// TIA Portal project "v6" (V15)

(* hardware
DEVICE "S7-1200 station_1"  S7-1200 Station
   slot 0: "Rack_0"  S7-1200 Rack  Rack  V1.0
   slot 1: "PLC_1"  CPU 1214C DC/DC/DC  6ES7 214-1AG40-0XB0  V4.2
*)

// ===== PLC "PLC_1"  CPU 1214C DC/DC/DC =====

VAR_GLOBAL   // PLC tag table "Default tag table"
   "truc1_Pulse" AT %Q0.3 : Bool;
   "truc1_Direction" AT %Q1.0 : Bool;
   "truc2_Pulse" AT %Q0.0 : Bool;
   "truc2_Direction" AT %Q0.1 : Bool;
   "truc3_Pulse" AT %Q0.4 : Bool;
   "truc3_Direction" AT %Q0.5 : Bool;
   "truc4_Pulse" AT %Q0.6 : Bool;
   "truc4_Direction" AT %Q0.7 : Bool;
   "Tag_1" AT %M0.0 : Bool;
   "Tag_2" AT %I0.0 : Bool;
   "Tag_3" AT %I0.3 : Bool;
   "vitricanden_truc1" AT %MD50 : Real;
   "kichtruc-1" AT %M1.0 : Bool;
   "Tag_6" AT %M5.0 : Bool;
   "vitricanden_truc2" AT %MD54 : Real;
   "kich_truc2" AT %M1.1 : Bool;
   "vitricanden_truc3" AT %MD58 : Real;
   "Tag_10" AT %M1.2 : Bool;
   "vitricanden_truc4" AT %MD62 : Real;
   "kich_truc4" AT %M1.3 : Bool;
   "Tag_13" AT %M5.1 : Bool;
   "Tag_14" AT %M5.2 : Bool;
   "Tag_15" AT %M5.3 : Bool;
   "Tag_16" AT %M10.0 : Bool;
   "Tag_17" AT %MW30 : Int;
   "goi vi tri" AT %M15.0 : Bool;
   "nhap vi tri goi" AT %MW32 : Int;
   "Tag_4" AT %I0.6 : Bool;
   "Tag_7" AT %I0.7 : Bool;
   "Tag_9" AT %I1.0 : Bool;
   "Tag_11" AT %I1.1 : Bool;
   "Tag_18" AT %I1.2 : Bool;
   "Tag_19" AT %I1.3 : Bool;
   "Tag_20" AT %I1.4 : Bool;
   "Tag_21" AT %I1.5 : Bool;
   "Tag_22" AT %M5.4 : Bool;
   "Tag_23" AT %M5.5 : Bool;
   "Tag_24" AT %M5.6 : Bool;
   "Tag_25" AT %M5.7 : Bool;
   "Tag_26" AT %M6.0 : Bool;
   "Tag_27" AT %M6.1 : Bool;
   "kich_truc_42" AT %M1.4 : Bool;
   "kich_truc_43" AT %M1.5 : Bool;
   "kich_truc_44" AT %M1.6 : Bool;
   "Tag_31" AT %M7.0 : Bool;
   "Tag_32" AT %M7.1 : Bool;
   "Tag_33" AT %M7.2 : Bool;
   "Tag_34" AT %M7.3 : Bool;
   "Tag_35" AT %M7.4 : Bool;
   "Tag_36" AT %M7.5 : Bool;
   "Tag_37" AT %M7.6 : Bool;
   "Tag_38" AT %M7.7 : Bool;
   "Tag_39" AT %M8.0 : Bool;
   "Tag_40" AT %M8.1 : Bool;
   "kich_truc1" AT %M2.0 : Bool;
   "kich_truc1(1)" AT %M2.1 : Bool;
   "kich_truc1(2)" AT %M2.2 : Bool;
   "kich_truc1(3)" AT %M2.3 : Bool;
   "kich_truc2(1)" AT %M2.4 : Bool;
   "kich_truc2(2)" AT %M2.5 : Bool;
   "kich_truc2(3)" AT %M2.6 : Bool;
   "kich_truc2(4)" AT %M2.7 : Bool;
   "kich_truc3(3)" AT %M3.0 : Bool;
   "kich_truc3(2)" AT %M3.1 : Bool;
   "kich_truc3" AT %M3.2 : Bool;
   "kich_truc3(1)" AT %M3.3 : Bool;
   "Tag_5" AT %M100.0 : Bool;
   "Tag_8" AT %M100.1 : Bool;
   "Tag_12" AT %M100.2 : Bool;
   "Tag_28" AT %M11.0 : Bool;
   "Tag_29" AT %M11.1 : Bool;
   "Tag_30" AT %M11.2 : Bool;
   "Tag_41" AT %M11.3 : Bool;
   "Tag_42" AT %M11.4 : Bool;
   "Tag_43" AT %M11.5 : Bool;
   "Tag_44" AT %M11.6 : Bool;
   "Tag_45" AT %M11.7 : Bool;
   "Tag_46" AT %M12.0 : Bool;
   "Tag_47" AT %M12.1 : Bool;
   "Tag_48" AT %M12.2 : Bool;
   "Tag_49" AT %M12.3 : Bool;
   "Tag_50" AT %M12.4 : Bool;
   "Tag_51" AT %M12.5 : Bool;
   "Tag_52" AT %M12.6 : Bool;
   "Tag_53" AT %M12.7 : Bool;
   "Tag_54" AT %M13.0 : Bool;
   "Tag_55" AT %M13.1 : Bool;
   "Tag_56" AT %M100.3 : Bool;
   "Tag_57" AT %M100.4 : Bool;
   "kich_truc_41" AT %M3.4 : Bool;
   "kich_truc3(4)" AT %M3.5 : Bool;
   "Kich_truc1_Home" AT %M3.6 : Bool;
   "Kich_truc2_Home" AT %M3.7 : Bool;
   "kich_truc3_Home" AT %M4.0 : Bool;
   "kich_truc4_Home" AT %M4.1 : Bool;
   "Tag_58" AT %M13.2 : Bool;
   "Tag_59" AT %M13.3 : Bool;
   "Tag_60" AT %M13.4 : Bool;
   "Tag_61" AT %M13.5 : Bool;
   "Tag_62" AT %M13.6 : Bool;
   "Tag_63" AT %M13.7 : Bool;
   "Tag_64" AT %M14.0 : Bool;
   "Tag_65" AT %M14.1 : Bool;
   "Tag_66" AT %M14.2 : Bool;
   "Tag_67" AT %M14.3 : Bool;
END_VAR

DATA_BLOCK "vitri"   // DB5
{ S7_Optimized_Access := 'FALSE' }
VERSION : 0.1
   VAR
      vitri4 : Array[0..3] of Real;
      vitri3 : Array[0..3] of Real;
      vitri2 : Array[0..3] of Real;
      Homing : Array[0..3] of Real;
      vitri1 : Array[0..3] of Real;
   END_VAR
BEGIN
END_DATA_BLOCK

DATA_BLOCK "tocdo"   // DB6
{ S7_Optimized_Access := 'FALSE' }
VERSION : 0.1
   VAR
      tocdo1 : Array[0..3] of Real;
   END_VAR
BEGIN
END_DATA_BLOCK

DATA_BLOCK "goi vitri_truc4"   // DB46
{ S7_Optimized_Access := 'TRUE' }
VERSION : 0.1
   VAR
      vitri1 : Array[0..4] of Bool;
   END_VAR
BEGIN
END_DATA_BLOCK

DATA_BLOCK "vitri_Homing"   // DB47
{ S7_Optimized_Access := 'TRUE' }
VERSION : 0.1
   VAR
      Home : Array[0..4] of Real;
   END_VAR
BEGIN
END_DATA_BLOCK

// folder: System blocks/Program resources

DATA_BLOCK "IEC_Timer_0_DB"   // DB23
{ S7_Optimized_Access := 'TRUE' }
AUTHOR : Simatic
FAMILY : IEC
NAME : IEC_TMR
VERSION : 1.0
// stored: InstanceOfName IEC_TIMER
"IEC_TIMER"
BEGIN
END_DATA_BLOCK

DATA_BLOCK "IEC_Timer_0_DB_1"   // DB24
{ S7_Optimized_Access := 'TRUE' }
AUTHOR : Simatic
FAMILY : IEC
NAME : IEC_TMR
VERSION : 1.0
// stored: InstanceOfName IEC_TIMER
"IEC_TIMER"
BEGIN
END_DATA_BLOCK

DATA_BLOCK "IEC_Timer_0_DB_2"   // DB25
{ S7_Optimized_Access := 'TRUE' }
AUTHOR : Simatic
FAMILY : IEC
NAME : IEC_TMR
VERSION : 1.0
// stored: InstanceOfName IEC_TIMER
"IEC_TIMER"
BEGIN
END_DATA_BLOCK

DATA_BLOCK "IEC_Timer_0_DB_3"   // DB26
{ S7_Optimized_Access := 'TRUE' }
AUTHOR : Simatic
FAMILY : IEC
NAME : IEC_TMR
VERSION : 1.0
// stored: InstanceOfName IEC_TIMER
"IEC_TIMER"
BEGIN
END_DATA_BLOCK

DATA_BLOCK "IEC_Timer_0_DB_4"   // DB27
{ S7_Optimized_Access := 'TRUE' }
AUTHOR : Simatic
FAMILY : IEC
NAME : IEC_TMR
VERSION : 1.0
// stored: InstanceOfName IEC_TIMER
"IEC_TIMER"
BEGIN
END_DATA_BLOCK

DATA_BLOCK "IEC_Timer_0_DB_5"   // DB28
{ S7_Optimized_Access := 'TRUE' }
AUTHOR : Simatic
FAMILY : IEC
NAME : IEC_TMR
VERSION : 1.0
// stored: InstanceOfName IEC_TIMER
"IEC_TIMER"
BEGIN
END_DATA_BLOCK

DATA_BLOCK "IEC_Timer_0_DB_6"   // DB29
{ S7_Optimized_Access := 'TRUE' }
AUTHOR : Simatic
FAMILY : IEC
NAME : IEC_TMR
VERSION : 1.0
// stored: InstanceOfName IEC_TIMER
"IEC_TIMER"
BEGIN
END_DATA_BLOCK

DATA_BLOCK "IEC_Timer_0_DB_7"   // DB30
{ S7_Optimized_Access := 'TRUE' }
AUTHOR : Simatic
FAMILY : IEC
NAME : IEC_TMR
VERSION : 1.0
// stored: InstanceOfName IEC_TIMER
"IEC_TIMER"
BEGIN
END_DATA_BLOCK

DATA_BLOCK "IEC_Timer_0_DB_8"   // DB31
{ S7_Optimized_Access := 'TRUE' }
AUTHOR : Simatic
FAMILY : IEC
NAME : IEC_TMR
VERSION : 1.0
// stored: InstanceOfName IEC_TIMER
"IEC_TIMER"
BEGIN
END_DATA_BLOCK

DATA_BLOCK "IEC_Timer_0_DB_9"   // DB32
{ S7_Optimized_Access := 'TRUE' }
AUTHOR : Simatic
FAMILY : IEC
NAME : IEC_TMR
VERSION : 1.0
// stored: InstanceOfName IEC_TIMER
"IEC_TIMER"
BEGIN
END_DATA_BLOCK

DATA_BLOCK "IEC_Timer_0_DB_10"   // DB33
{ S7_Optimized_Access := 'TRUE' }
AUTHOR : Simatic
FAMILY : IEC
NAME : IEC_TMR
VERSION : 1.0
// stored: InstanceOfName IEC_TIMER
"IEC_TIMER"
BEGIN
END_DATA_BLOCK

DATA_BLOCK "IEC_Timer_0_DB_11"   // DB34
{ S7_Optimized_Access := 'TRUE' }
AUTHOR : Simatic
FAMILY : IEC
NAME : IEC_TMR
VERSION : 1.0
// stored: InstanceOfName IEC_TIMER
"IEC_TIMER"
BEGIN
END_DATA_BLOCK

DATA_BLOCK "IEC_Timer_0_DB_12"   // DB35
{ S7_Optimized_Access := 'TRUE' }
AUTHOR : Simatic
FAMILY : IEC
NAME : IEC_TMR
VERSION : 1.0
// stored: InstanceOfName IEC_TIMER
"IEC_TIMER"
BEGIN
END_DATA_BLOCK

DATA_BLOCK "IEC_Timer_0_DB_13"   // DB36
{ S7_Optimized_Access := 'TRUE' }
AUTHOR : Simatic
FAMILY : IEC
NAME : IEC_TMR
VERSION : 1.0
// stored: InstanceOfName IEC_TIMER
"IEC_TIMER"
BEGIN
END_DATA_BLOCK

DATA_BLOCK "IEC_Timer_0_DB_14"   // DB37
{ S7_Optimized_Access := 'TRUE' }
AUTHOR : Simatic
FAMILY : IEC
NAME : IEC_TMR
VERSION : 1.0
// stored: InstanceOfName IEC_TIMER
"IEC_TIMER"
BEGIN
END_DATA_BLOCK

DATA_BLOCK "IEC_Timer_0_DB_15"   // DB38
{ S7_Optimized_Access := 'TRUE' }
AUTHOR : Simatic
FAMILY : IEC
NAME : IEC_TMR
VERSION : 1.0
// stored: InstanceOfName IEC_TIMER
"IEC_TIMER"
BEGIN
END_DATA_BLOCK

DATA_BLOCK "IEC_Timer_0_DB_16"   // DB39
{ S7_Optimized_Access := 'TRUE' }
AUTHOR : Simatic
FAMILY : IEC
NAME : IEC_TMR
VERSION : 1.0
// stored: InstanceOfName IEC_TIMER
"IEC_TIMER"
BEGIN
END_DATA_BLOCK

DATA_BLOCK "IEC_Timer_0_DB_17"   // DB40
{ S7_Optimized_Access := 'TRUE' }
AUTHOR : Simatic
FAMILY : IEC
NAME : IEC_TMR
VERSION : 1.0
// stored: InstanceOfName IEC_TIMER
"IEC_TIMER"
BEGIN
END_DATA_BLOCK

DATA_BLOCK "IEC_Timer_0_DB_18"   // DB41
{ S7_Optimized_Access := 'TRUE' }
AUTHOR : Simatic
FAMILY : IEC
NAME : IEC_TMR
VERSION : 1.0
// stored: InstanceOfName IEC_TIMER
"IEC_TIMER"
BEGIN
END_DATA_BLOCK

DATA_BLOCK "IEC_Timer_0_DB_19"   // DB42
{ S7_Optimized_Access := 'TRUE' }
AUTHOR : Simatic
FAMILY : IEC
NAME : IEC_TMR
VERSION : 1.0
// stored: InstanceOfName IEC_TIMER
"IEC_TIMER"
BEGIN
END_DATA_BLOCK

DATA_BLOCK "IEC_Timer_0_DB_20"   // DB43
{ S7_Optimized_Access := 'TRUE' }
AUTHOR : Simatic
FAMILY : IEC
NAME : IEC_TMR
VERSION : 1.0
// stored: InstanceOfName IEC_TIMER
"IEC_TIMER"
BEGIN
END_DATA_BLOCK

DATA_BLOCK "IEC_Timer_0_DB_21"   // DB44
{ S7_Optimized_Access := 'TRUE' }
AUTHOR : Simatic
FAMILY : IEC
NAME : IEC_TMR
VERSION : 1.0
// stored: InstanceOfName IEC_TIMER
"IEC_TIMER"
BEGIN
END_DATA_BLOCK

DATA_BLOCK "IEC_Timer_0_DB_22"   // DB45
{ S7_Optimized_Access := 'TRUE' }
AUTHOR : Simatic
FAMILY : IEC
NAME : IEC_TMR
VERSION : 1.0
// stored: InstanceOfName IEC_TIMER
"IEC_TIMER"
BEGIN
END_DATA_BLOCK

DATA_BLOCK "IEC_Timer_0_DB_23"   // DB48
{ S7_Optimized_Access := 'TRUE' }
AUTHOR : Simatic
FAMILY : IEC
NAME : IEC_TMR
VERSION : 1.0
// stored: InstanceOfName IEC_TIMER
"IEC_TIMER"
BEGIN
END_DATA_BLOCK

DATA_BLOCK "IEC_Timer_0_DB_24"   // DB49
{ S7_Optimized_Access := 'TRUE' }
AUTHOR : Simatic
FAMILY : IEC
NAME : IEC_TMR
VERSION : 1.0
// stored: InstanceOfName IEC_TIMER
"IEC_TIMER"
BEGIN
END_DATA_BLOCK

DATA_BLOCK "IEC_Timer_0_DB_25"   // DB50
{ S7_Optimized_Access := 'TRUE' }
AUTHOR : Simatic
FAMILY : IEC
NAME : IEC_TMR
VERSION : 1.0
// stored: InstanceOfName IEC_TIMER
"IEC_TIMER"
BEGIN
END_DATA_BLOCK

DATA_BLOCK "IEC_Timer_0_DB_26"   // DB51
{ S7_Optimized_Access := 'TRUE' }
AUTHOR : Simatic
FAMILY : IEC
NAME : IEC_TMR
VERSION : 1.0
// stored: InstanceOfName IEC_TIMER
"IEC_TIMER"
BEGIN
END_DATA_BLOCK

// folder: (top level)

DATA_BLOCK "truc1"   // DB1, Motion_DB
{ S7_Optimized_Access := 'TRUE' }
AUTHOR : SIMATIC
FAMILY : BasicMC
NAME : TO_PosAx
VERSION : 6.0
// stored: InstanceOfName TO_PositioningAxis
"TO_PositioningAxis"
BEGIN
   // Axis.DirectionOutputEnabledCU = TRUE
   // Axis.OnlinePtoModeCU = 16#0000_0002
   // Axis.SelectedChannel2EnumCU = %Q1.0
   // Axis.SelectedChannel1EnumCU = %Q0.3
   // Pulse.MinDeltaDeltaFrequencyCU = 0.004
   // Pulse.MaxDeltaDeltaFrequencyCU = 1.0E+10
   // Pulse.MinDeltaFrequencyCU = 0.005
   // Pulse.MaxDeltaFrequencyCU = 9.5E+9
   // Pulse.MinFrequencyCU = 1.0
   // Pulse.MaxFrequencyCU = 100000.0
   // Pulse.OutputSourceCU = 16#0000_0000
   // Axis.SelectPTO = 1
   // Axis.OnlinePtoIndexCU = 1
END_DATA_BLOCK

DATA_BLOCK "truc2"   // DB2, Motion_DB
{ S7_Optimized_Access := 'TRUE' }
AUTHOR : SIMATIC
FAMILY : BasicMC
NAME : TO_PosAx
VERSION : 6.0
// stored: InstanceOfName TO_PositioningAxis
"TO_PositioningAxis"
BEGIN
   // Axis.DirectionOutputEnabledCU = TRUE
   // Axis.OnlinePtoModeCU = 16#0000_0002
   // Axis.SelectedChannel2EnumCU = %Q0.1
   // Axis.SelectedChannel1EnumCU = %Q0.0
   // Pulse.MinDeltaDeltaFrequencyCU = 0.004
   // Pulse.MaxDeltaDeltaFrequencyCU = 1.0E+10
   // Pulse.MinDeltaFrequencyCU = 0.005
   // Pulse.MaxDeltaFrequencyCU = 9.5E+9
   // Pulse.MinFrequencyCU = 1.0
   // Pulse.MaxFrequencyCU = 100000.0
   // Pulse.OutputSourceCU = 16#0000_0000
   // Axis.SelectPTO = 0
END_DATA_BLOCK

DATA_BLOCK "truc3"   // DB3, Motion_DB
{ S7_Optimized_Access := 'TRUE' }
AUTHOR : SIMATIC
FAMILY : BasicMC
NAME : TO_PosAx
VERSION : 6.0
// stored: InstanceOfName TO_PositioningAxis
"TO_PositioningAxis"
BEGIN
   // Axis.DirectionOutputEnabledCU = TRUE
   // Axis.OnlinePtoModeCU = 16#0000_0002
   // Axis.SelectedChannel2EnumCU = %Q0.5
   // Axis.SelectedChannel1EnumCU = %Q0.4
   // Pulse.MinDeltaDeltaFrequencyCU = 0.004
   // Pulse.MaxDeltaDeltaFrequencyCU = 1.0E+10
   // Pulse.MinDeltaFrequencyCU = 0.005
   // Pulse.MaxDeltaFrequencyCU = 9.5E+9
   // Pulse.MinFrequencyCU = 1.0
   // Pulse.MaxFrequencyCU = 30000.0
   // Pulse.OutputSourceCU = 16#0000_0000
   // Axis.SelectPTO = 2
   // Axis.OnlinePtoIndexCU = 2
END_DATA_BLOCK

DATA_BLOCK "truc4"   // DB4, Motion_DB
{ S7_Optimized_Access := 'TRUE' }
AUTHOR : SIMATIC
FAMILY : BasicMC
NAME : TO_PosAx
VERSION : 6.0
// stored: InstanceOfName TO_PositioningAxis
"TO_PositioningAxis"
BEGIN
   // Axis.DirectionOutputEnabledCU = TRUE
   // Axis.OnlinePtoModeCU = 16#0000_0002
   // Axis.SelectedChannel2EnumCU = %Q0.7
   // Axis.SelectedChannel1EnumCU = %Q0.6
   // Pulse.MinDeltaDeltaFrequencyCU = 0.004
   // Pulse.MaxDeltaDeltaFrequencyCU = 1.0E+10
   // Pulse.MinDeltaFrequencyCU = 0.005
   // Pulse.MaxDeltaFrequencyCU = 9.5E+9
   // Pulse.MinFrequencyCU = 1.0
   // Pulse.MaxFrequencyCU = 30000.0
   // Pulse.OutputSourceCU = 16#0000_0000
   // Axis.SelectPTO = 3
   // Axis.OnlinePtoIndexCU = 3
END_DATA_BLOCK

FUNCTION "configure_initial" : Void   // FC1, LAD
{ S7_Optimized_Access := 'TRUE' }
VERSION : 0.1
BEGIN

REGION Network 1
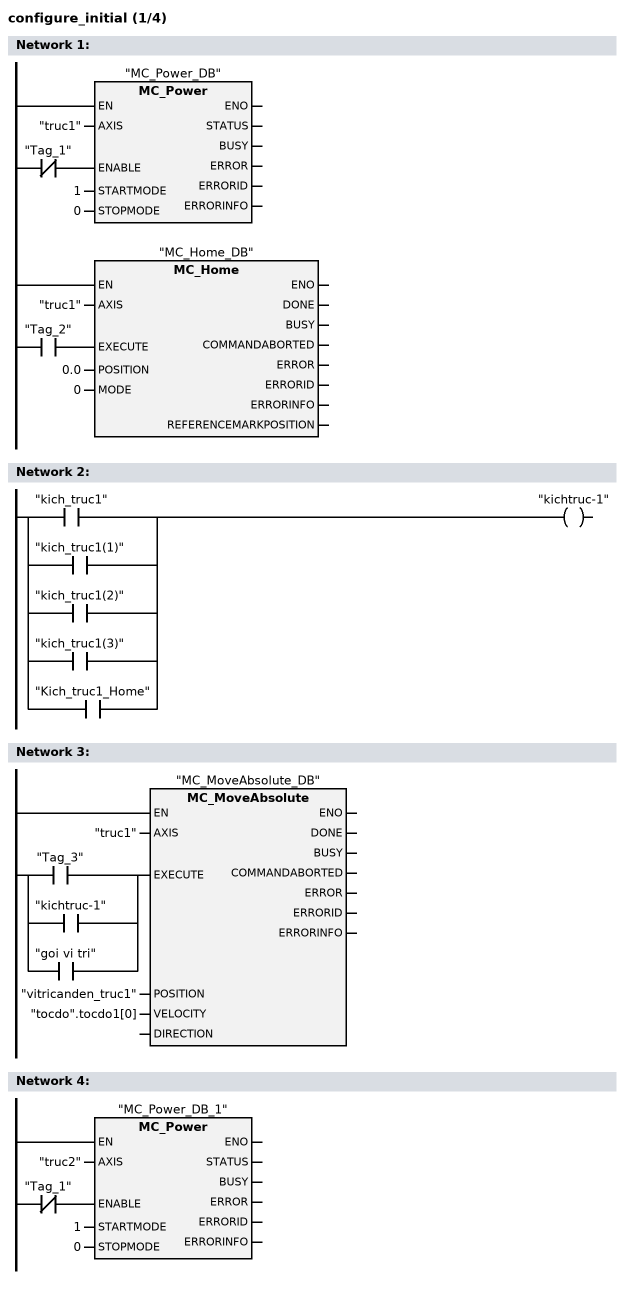
   "MC_Power_DB"(Axis := "truc1", Enable := NOT "Tag_1", StartMode := 1, StopMode := 0);   // MC_Power
   "MC_Home_DB"(Axis := "truc1", Execute := "Tag_2", Position := 0.0, Mode := 0);   // MC_Home
END_REGION

REGION Network 2
   RUNG wire#powerrail
      Contact( "kich_truc1" )
      wire#w1
      Coil( "kichtruc-1" )
   END_RUNG
   RUNG wire#powerrail
      Contact( "kich_truc1(1)" )
   END_RUNG wire#w1
   RUNG wire#powerrail
      Contact( "kich_truc1(2)" )
   END_RUNG wire#w1
   RUNG wire#powerrail
      Contact( "kich_truc1(3)" )
   END_RUNG wire#w1
   RUNG wire#powerrail
      Contact( "Kich_truc1_Home" )
   END_RUNG wire#w1
   // the same network as SCL:
   "kichtruc-1" := "kich_truc1" OR "kich_truc1(1)" OR "kich_truc1(2)" OR "kich_truc1(3)" OR "Kich_truc1_Home";
END_REGION

REGION Network 3
   "MC_MoveAbsolute_DB"(Axis := "truc1",   // MC_MoveAbsolute
                        Execute := "Tag_3" OR "kichtruc-1" OR "goi vi tri",
                        Position := "vitricanden_truc1",
                        Velocity := "tocdo".tocdo1[0]);
END_REGION

REGION Network 4
   "MC_Power_DB_1"(Axis := "truc2", Enable := NOT "Tag_1", StartMode := 1, StopMode := 0);   // MC_Power
END_REGION

REGION Network 5
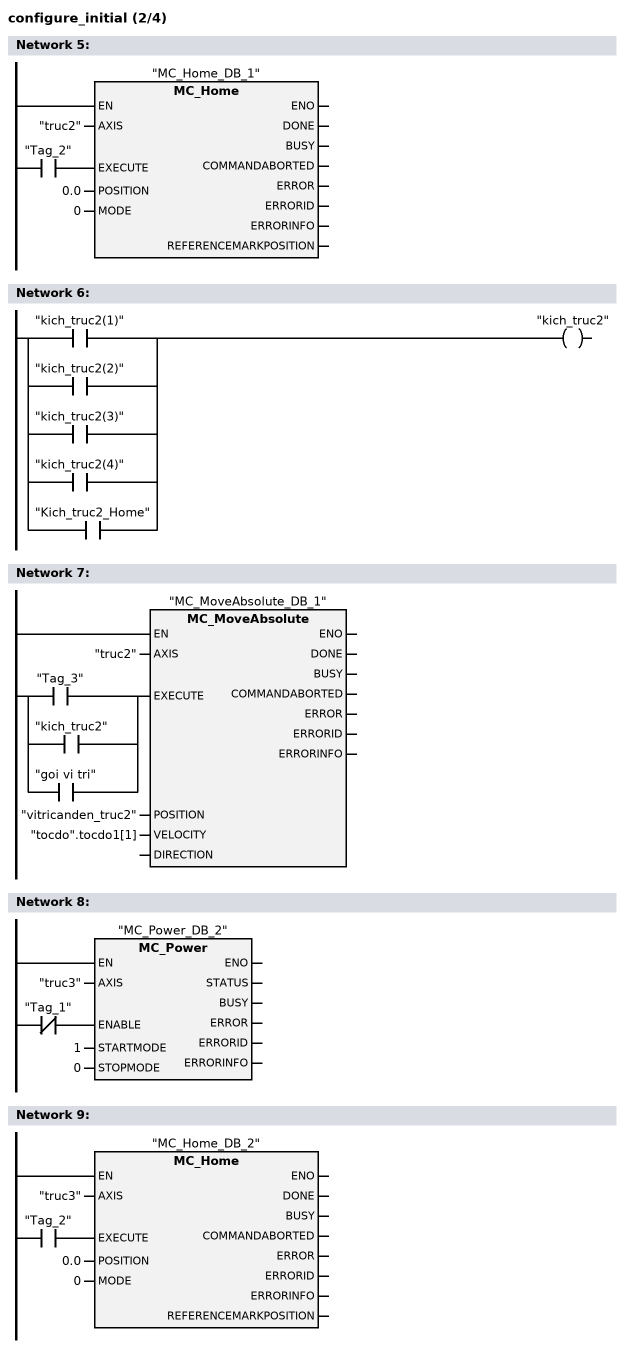
   "MC_Home_DB_1"(Axis := "truc2", Execute := "Tag_2", Position := 0.0, Mode := 0);   // MC_Home
END_REGION

REGION Network 6
   RUNG wire#powerrail
      Contact( "kich_truc2(1)" )
      wire#w1
      Coil( "kich_truc2" )
   END_RUNG
   RUNG wire#powerrail
      Contact( "kich_truc2(2)" )
   END_RUNG wire#w1
   RUNG wire#powerrail
      Contact( "kich_truc2(3)" )
   END_RUNG wire#w1
   RUNG wire#powerrail
      Contact( "kich_truc2(4)" )
   END_RUNG wire#w1
   RUNG wire#powerrail
      Contact( "Kich_truc2_Home" )
   END_RUNG wire#w1
   // the same network as SCL:
   "kich_truc2" := "kich_truc2(1)" OR "kich_truc2(2)" OR "kich_truc2(3)" OR "kich_truc2(4)" OR "Kich_truc2_Home";
END_REGION

REGION Network 7
   "MC_MoveAbsolute_DB_1"(Axis := "truc2",   // MC_MoveAbsolute
                          Execute := "Tag_3" OR "kich_truc2" OR "goi vi tri",
                          Position := "vitricanden_truc2",
                          Velocity := "tocdo".tocdo1[1]);
END_REGION

REGION Network 8
   "MC_Power_DB_2"(Axis := "truc3", Enable := NOT "Tag_1", StartMode := 1, StopMode := 0);   // MC_Power
END_REGION

REGION Network 9
   "MC_Home_DB_2"(Axis := "truc3", Execute := "Tag_2", Position := 0.0, Mode := 0);   // MC_Home
END_REGION

REGION Network 10
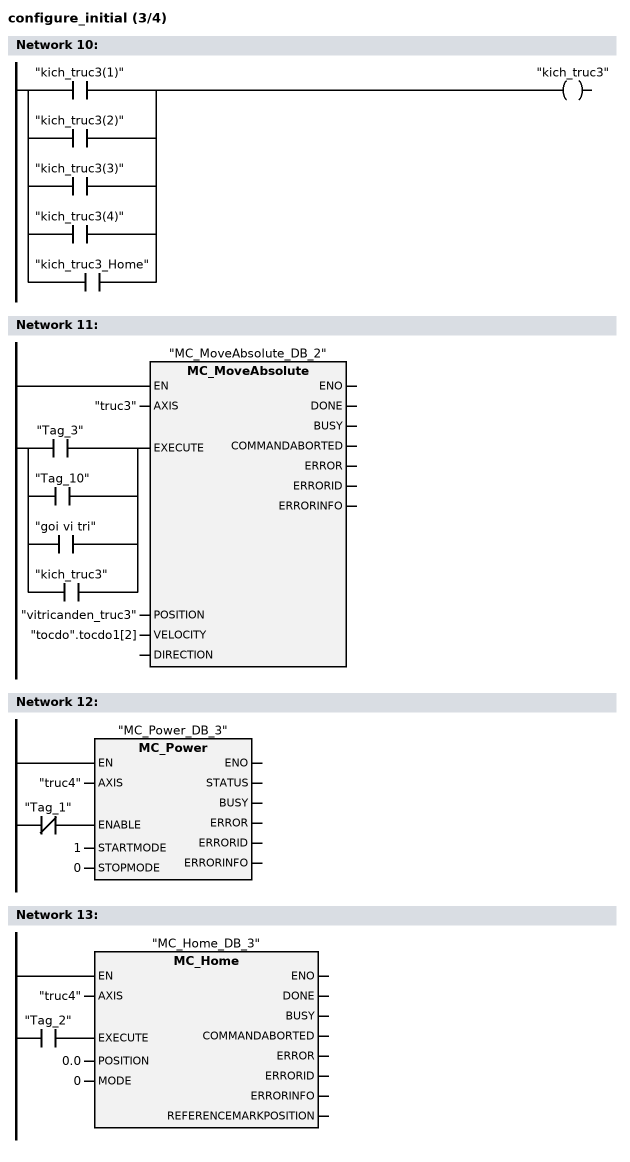
   RUNG wire#powerrail
      Contact( "kich_truc3(1)" )
      wire#w1
      Coil( "kich_truc3" )
   END_RUNG
   RUNG wire#powerrail
      Contact( "kich_truc3(2)" )
   END_RUNG wire#w1
   RUNG wire#powerrail
      Contact( "kich_truc3(3)" )
   END_RUNG wire#w1
   RUNG wire#powerrail
      Contact( "kich_truc3(4)" )
   END_RUNG wire#w1
   RUNG wire#powerrail
      Contact( "kich_truc3_Home" )
   END_RUNG wire#w1
   // the same network as SCL:
   "kich_truc3" := "kich_truc3(1)" OR "kich_truc3(2)" OR "kich_truc3(3)" OR "kich_truc3(4)" OR "kich_truc3_Home";
END_REGION

REGION Network 11
   "MC_MoveAbsolute_DB_2"(Axis := "truc3",   // MC_MoveAbsolute
                          Execute := "Tag_3" OR "Tag_10" OR "goi vi tri" OR "kich_truc3",
                          Position := "vitricanden_truc3",
                          Velocity := "tocdo".tocdo1[2]);
END_REGION

REGION Network 12
   "MC_Power_DB_3"(Axis := "truc4", Enable := NOT "Tag_1", StartMode := 1, StopMode := 0);   // MC_Power
END_REGION

REGION Network 13
   "MC_Home_DB_3"(Axis := "truc4", Execute := "Tag_2", Position := 0.0, Mode := 0);   // MC_Home
END_REGION

REGION Network 14
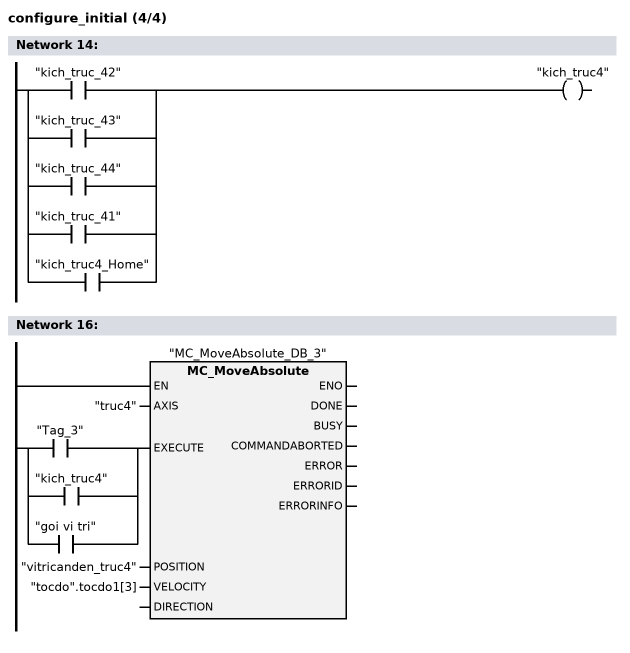
   RUNG wire#powerrail
      Contact( "kich_truc_42" )
      wire#w1
      Coil( "kich_truc4" )
   END_RUNG
   RUNG wire#powerrail
      Contact( "kich_truc_43" )
   END_RUNG wire#w1
   RUNG wire#powerrail
      Contact( "kich_truc_44" )
   END_RUNG wire#w1
   RUNG wire#powerrail
      Contact( "kich_truc_41" )
   END_RUNG wire#w1
   RUNG wire#powerrail
      Contact( "kich_truc4_Home" )
   END_RUNG wire#w1
   // the same network as SCL:
   "kich_truc4" := "kich_truc_42" OR "kich_truc_43" OR "kich_truc_44" OR "kich_truc_41" OR "kich_truc4_Home";
END_REGION

REGION Network 16
   "MC_MoveAbsolute_DB_3"(Axis := "truc4",   // MC_MoveAbsolute
                          Execute := "Tag_3" OR "kich_truc4" OR "goi vi tri",
                          Position := "vitricanden_truc4",
                          Velocity := "tocdo".tocdo1[3]);
END_REGION
END_FUNCTION

FUNCTION "luuvitri" : Void   // FC2, LAD
{ S7_Optimized_Access := 'TRUE' }
VERSION : 0.1
BEGIN

REGION Network 1
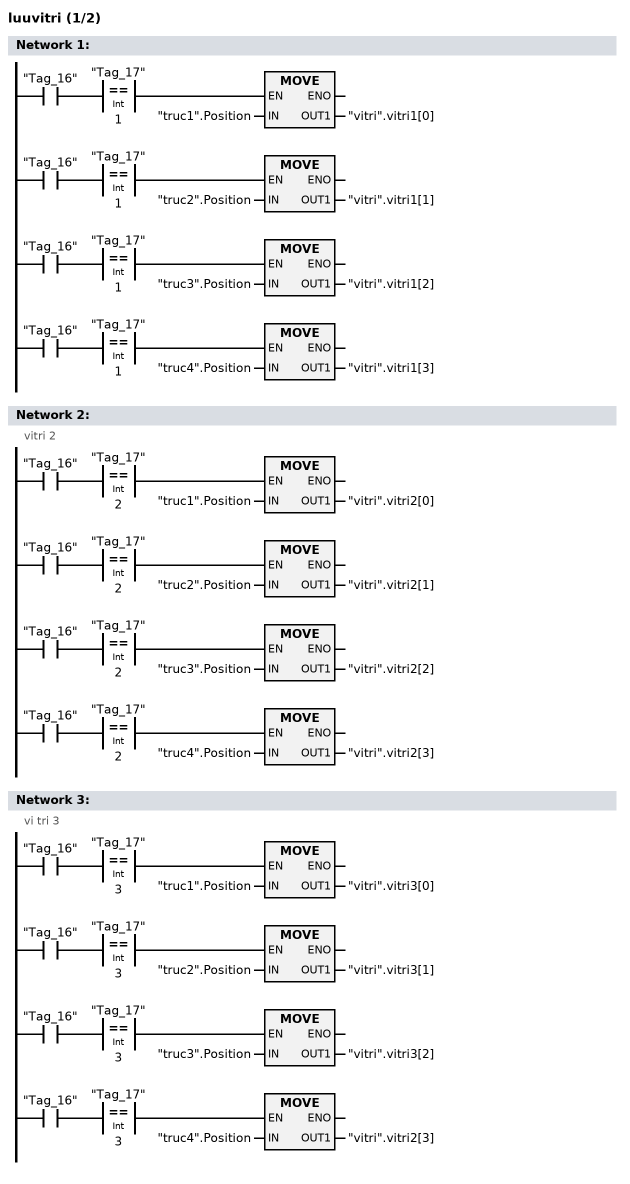
   RUNG wire#powerrail
      Contact( "Tag_16" )
      { S7_Templates := "SrcType := Int" } EQ_Contact(in1 := "Tag_17", in2 := 1)
      Move(in := "truc1".Position, out1 => "vitri".vitri1[0])
   END_RUNG
   RUNG wire#powerrail
      Contact( "Tag_16" )
      { S7_Templates := "SrcType := Int" } EQ_Contact(in1 := "Tag_17", in2 := 1)
      Move(in := "truc2".Position, out1 => "vitri".vitri1[1])
   END_RUNG
   RUNG wire#powerrail
      Contact( "Tag_16" )
      { S7_Templates := "SrcType := Int" } EQ_Contact(in1 := "Tag_17", in2 := 1)
      Move(in := "truc3".Position, out1 => "vitri".vitri1[2])
   END_RUNG
   RUNG wire#powerrail
      Contact( "Tag_16" )
      { S7_Templates := "SrcType := Int" } EQ_Contact(in1 := "Tag_17", in2 := 1)
      Move(in := "truc4".Position, out1 => "vitri".vitri1[3])
   END_RUNG
   // the same network as SCL:
   IF "Tag_16" AND ("Tag_17" = 1) THEN
       "vitri".vitri1[0] := "truc1".Position;
       "vitri".vitri1[1] := "truc2".Position;
       "vitri".vitri1[2] := "truc3".Position;
       "vitri".vitri1[3] := "truc4".Position;
   END_IF;
END_REGION

REGION Network 2
   // vitri 2
   RUNG wire#powerrail
      Contact( "Tag_16" )
      { S7_Templates := "SrcType := Int" } EQ_Contact(in1 := "Tag_17", in2 := 2)
      Move(in := "truc1".Position, out1 => "vitri".vitri2[0])
   END_RUNG
   RUNG wire#powerrail
      Contact( "Tag_16" )
      { S7_Templates := "SrcType := Int" } EQ_Contact(in1 := "Tag_17", in2 := 2)
      Move(in := "truc2".Position, out1 => "vitri".vitri2[1])
   END_RUNG
   RUNG wire#powerrail
      Contact( "Tag_16" )
      { S7_Templates := "SrcType := Int" } EQ_Contact(in1 := "Tag_17", in2 := 2)
      Move(in := "truc3".Position, out1 => "vitri".vitri2[2])
   END_RUNG
   RUNG wire#powerrail
      Contact( "Tag_16" )
      { S7_Templates := "SrcType := Int" } EQ_Contact(in1 := "Tag_17", in2 := 2)
      Move(in := "truc4".Position, out1 => "vitri".vitri2[3])
   END_RUNG
   // the same network as SCL:
   IF "Tag_16" AND ("Tag_17" = 2) THEN
       "vitri".vitri2[0] := "truc1".Position;
       "vitri".vitri2[1] := "truc2".Position;
       "vitri".vitri2[2] := "truc3".Position;
       "vitri".vitri2[3] := "truc4".Position;
   END_IF;
END_REGION

REGION Network 3
   // vi tri 3
   RUNG wire#powerrail
      Contact( "Tag_16" )
      { S7_Templates := "SrcType := Int" } EQ_Contact(in1 := "Tag_17", in2 := 3)
      Move(in := "truc1".Position, out1 => "vitri".vitri3[0])
   END_RUNG
   RUNG wire#powerrail
      Contact( "Tag_16" )
      { S7_Templates := "SrcType := Int" } EQ_Contact(in1 := "Tag_17", in2 := 3)
      Move(in := "truc2".Position, out1 => "vitri".vitri3[1])
   END_RUNG
   RUNG wire#powerrail
      Contact( "Tag_16" )
      { S7_Templates := "SrcType := Int" } EQ_Contact(in1 := "Tag_17", in2 := 3)
      Move(in := "truc3".Position, out1 => "vitri".vitri3[2])
   END_RUNG
   RUNG wire#powerrail
      Contact( "Tag_16" )
      { S7_Templates := "SrcType := Int" } EQ_Contact(in1 := "Tag_17", in2 := 3)
      Move(in := "truc4".Position, out1 => "vitri".vitri2[3])
   END_RUNG
   // the same network as SCL:
   IF "Tag_16" AND ("Tag_17" = 3) THEN
       "vitri".vitri3[0] := "truc1".Position;
       "vitri".vitri3[1] := "truc2".Position;
       "vitri".vitri3[2] := "truc3".Position;
       "vitri".vitri2[3] := "truc4".Position;
   END_IF;
END_REGION

REGION Network 4
   // vi tri 3
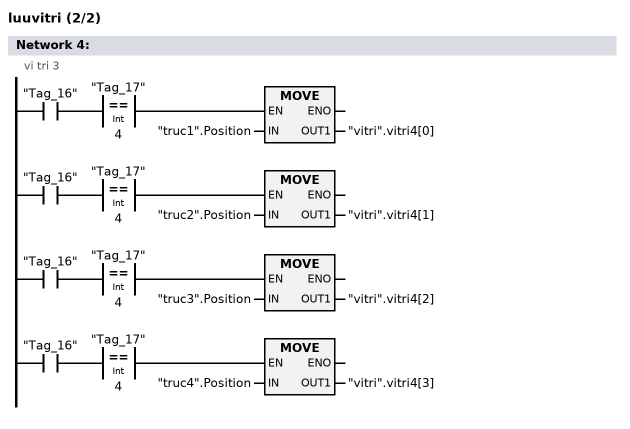
   RUNG wire#powerrail
      Contact( "Tag_16" )
      { S7_Templates := "SrcType := Int" } EQ_Contact(in1 := "Tag_17", in2 := 4)
      Move(in := "truc1".Position, out1 => "vitri".vitri4[0])
   END_RUNG
   RUNG wire#powerrail
      Contact( "Tag_16" )
      { S7_Templates := "SrcType := Int" } EQ_Contact(in1 := "Tag_17", in2 := 4)
      Move(in := "truc2".Position, out1 => "vitri".vitri4[1])
   END_RUNG
   RUNG wire#powerrail
      Contact( "Tag_16" )
      { S7_Templates := "SrcType := Int" } EQ_Contact(in1 := "Tag_17", in2 := 4)
      Move(in := "truc3".Position, out1 => "vitri".vitri4[2])
   END_RUNG
   RUNG wire#powerrail
      Contact( "Tag_16" )
      { S7_Templates := "SrcType := Int" } EQ_Contact(in1 := "Tag_17", in2 := 4)
      Move(in := "truc4".Position, out1 => "vitri".vitri4[3])
   END_RUNG
   // the same network as SCL:
   IF "Tag_16" AND ("Tag_17" = 4) THEN
       "vitri".vitri4[0] := "truc1".Position;
       "vitri".vitri4[1] := "truc2".Position;
       "vitri".vitri4[2] := "truc3".Position;
       "vitri".vitri4[3] := "truc4".Position;
   END_IF;
END_REGION
END_FUNCTION

FUNCTION "goivitri" : Void   // FC3, LAD
{ S7_Optimized_Access := 'TRUE' }
VERSION : 0.1
BEGIN

REGION Network 1
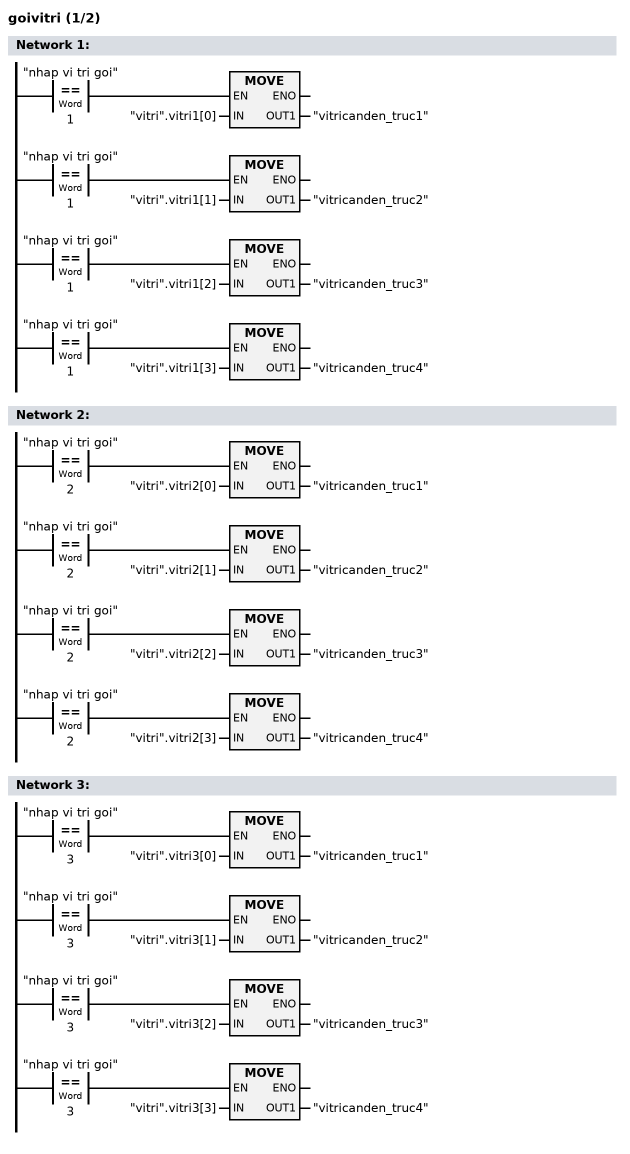
   RUNG wire#powerrail
      { S7_Templates := "SrcType := Word" } EQ_Contact(in1 := "nhap vi tri goi", in2 := 1)
      Move(in := "vitri".vitri1[0], out1 => "vitricanden_truc1")
   END_RUNG
   RUNG wire#powerrail
      { S7_Templates := "SrcType := Word" } EQ_Contact(in1 := "nhap vi tri goi", in2 := 1)
      Move(in := "vitri".vitri1[1], out1 => "vitricanden_truc2")
   END_RUNG
   RUNG wire#powerrail
      { S7_Templates := "SrcType := Word" } EQ_Contact(in1 := "nhap vi tri goi", in2 := 1)
      Move(in := "vitri".vitri1[2], out1 => "vitricanden_truc3")
   END_RUNG
   RUNG wire#powerrail
      { S7_Templates := "SrcType := Word" } EQ_Contact(in1 := "nhap vi tri goi", in2 := 1)
      Move(in := "vitri".vitri1[3], out1 => "vitricanden_truc4")
   END_RUNG
   // the same network as SCL:
   IF "nhap vi tri goi" = 1 THEN
       "vitricanden_truc1" := "vitri".vitri1[0];
       "vitricanden_truc2" := "vitri".vitri1[1];
       "vitricanden_truc3" := "vitri".vitri1[2];
       "vitricanden_truc4" := "vitri".vitri1[3];
   END_IF;
END_REGION

REGION Network 2
   RUNG wire#powerrail
      { S7_Templates := "SrcType := Word" } EQ_Contact(in1 := "nhap vi tri goi", in2 := 2)
      Move(in := "vitri".vitri2[0], out1 => "vitricanden_truc1")
   END_RUNG
   RUNG wire#powerrail
      { S7_Templates := "SrcType := Word" } EQ_Contact(in1 := "nhap vi tri goi", in2 := 2)
      Move(in := "vitri".vitri2[1], out1 => "vitricanden_truc2")
   END_RUNG
   RUNG wire#powerrail
      { S7_Templates := "SrcType := Word" } EQ_Contact(in1 := "nhap vi tri goi", in2 := 2)
      Move(in := "vitri".vitri2[2], out1 => "vitricanden_truc3")
   END_RUNG
   RUNG wire#powerrail
      { S7_Templates := "SrcType := Word" } EQ_Contact(in1 := "nhap vi tri goi", in2 := 2)
      Move(in := "vitri".vitri2[3], out1 => "vitricanden_truc4")
   END_RUNG
   // the same network as SCL:
   IF "nhap vi tri goi" = 2 THEN
       "vitricanden_truc1" := "vitri".vitri2[0];
       "vitricanden_truc2" := "vitri".vitri2[1];
       "vitricanden_truc3" := "vitri".vitri2[2];
       "vitricanden_truc4" := "vitri".vitri2[3];
   END_IF;
END_REGION

REGION Network 3
   RUNG wire#powerrail
      { S7_Templates := "SrcType := Word" } EQ_Contact(in1 := "nhap vi tri goi", in2 := 3)
      Move(in := "vitri".vitri3[0], out1 => "vitricanden_truc1")
   END_RUNG
   RUNG wire#powerrail
      { S7_Templates := "SrcType := Word" } EQ_Contact(in1 := "nhap vi tri goi", in2 := 3)
      Move(in := "vitri".vitri3[1], out1 => "vitricanden_truc2")
   END_RUNG
   RUNG wire#powerrail
      { S7_Templates := "SrcType := Word" } EQ_Contact(in1 := "nhap vi tri goi", in2 := 3)
      Move(in := "vitri".vitri3[2], out1 => "vitricanden_truc3")
   END_RUNG
   RUNG wire#powerrail
      { S7_Templates := "SrcType := Word" } EQ_Contact(in1 := "nhap vi tri goi", in2 := 3)
      Move(in := "vitri".vitri3[3], out1 => "vitricanden_truc4")
   END_RUNG
   // the same network as SCL:
   IF "nhap vi tri goi" = 3 THEN
       "vitricanden_truc1" := "vitri".vitri3[0];
       "vitricanden_truc2" := "vitri".vitri3[1];
       "vitricanden_truc3" := "vitri".vitri3[2];
       "vitricanden_truc4" := "vitri".vitri3[3];
   END_IF;
END_REGION

REGION Network 4
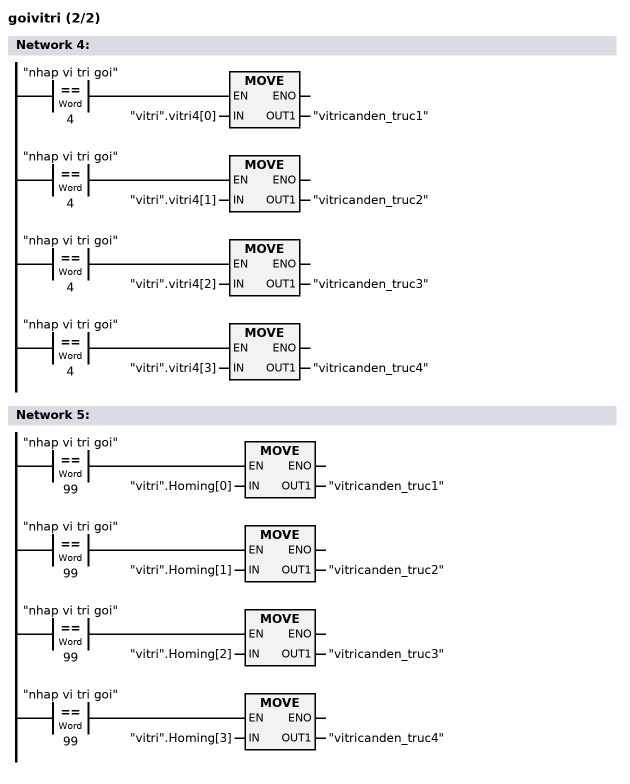
   RUNG wire#powerrail
      { S7_Templates := "SrcType := Word" } EQ_Contact(in1 := "nhap vi tri goi", in2 := 4)
      Move(in := "vitri".vitri4[0], out1 => "vitricanden_truc1")
   END_RUNG
   RUNG wire#powerrail
      { S7_Templates := "SrcType := Word" } EQ_Contact(in1 := "nhap vi tri goi", in2 := 4)
      Move(in := "vitri".vitri4[1], out1 => "vitricanden_truc2")
   END_RUNG
   RUNG wire#powerrail
      { S7_Templates := "SrcType := Word" } EQ_Contact(in1 := "nhap vi tri goi", in2 := 4)
      Move(in := "vitri".vitri4[2], out1 => "vitricanden_truc3")
   END_RUNG
   RUNG wire#powerrail
      { S7_Templates := "SrcType := Word" } EQ_Contact(in1 := "nhap vi tri goi", in2 := 4)
      Move(in := "vitri".vitri4[3], out1 => "vitricanden_truc4")
   END_RUNG
   // the same network as SCL:
   IF "nhap vi tri goi" = 4 THEN
       "vitricanden_truc1" := "vitri".vitri4[0];
       "vitricanden_truc2" := "vitri".vitri4[1];
       "vitricanden_truc3" := "vitri".vitri4[2];
       "vitricanden_truc4" := "vitri".vitri4[3];
   END_IF;
END_REGION

REGION Network 5
   RUNG wire#powerrail
      { S7_Templates := "SrcType := Word" } EQ_Contact(in1 := "nhap vi tri goi", in2 := 99)
      Move(in := "vitri".Homing[0], out1 => "vitricanden_truc1")
   END_RUNG
   RUNG wire#powerrail
      { S7_Templates := "SrcType := Word" } EQ_Contact(in1 := "nhap vi tri goi", in2 := 99)
      Move(in := "vitri".Homing[1], out1 => "vitricanden_truc2")
   END_RUNG
   RUNG wire#powerrail
      { S7_Templates := "SrcType := Word" } EQ_Contact(in1 := "nhap vi tri goi", in2 := 99)
      Move(in := "vitri".Homing[2], out1 => "vitricanden_truc3")
   END_RUNG
   RUNG wire#powerrail
      { S7_Templates := "SrcType := Word" } EQ_Contact(in1 := "nhap vi tri goi", in2 := 99)
      Move(in := "vitri".Homing[3], out1 => "vitricanden_truc4")
   END_RUNG
   // the same network as SCL:
   IF "nhap vi tri goi" = 99 THEN
       "vitricanden_truc1" := "vitri".Homing[0];
       "vitricanden_truc2" := "vitri".Homing[1];
       "vitricanden_truc3" := "vitri".Homing[2];
       "vitricanden_truc4" := "vitri".Homing[3];
   END_IF;
END_REGION
END_FUNCTION

FUNCTION "Run_Job" : Void   // FC4, LAD
{ S7_Optimized_Access := 'TRUE' }
VERSION : 0.1
BEGIN

REGION Network 1
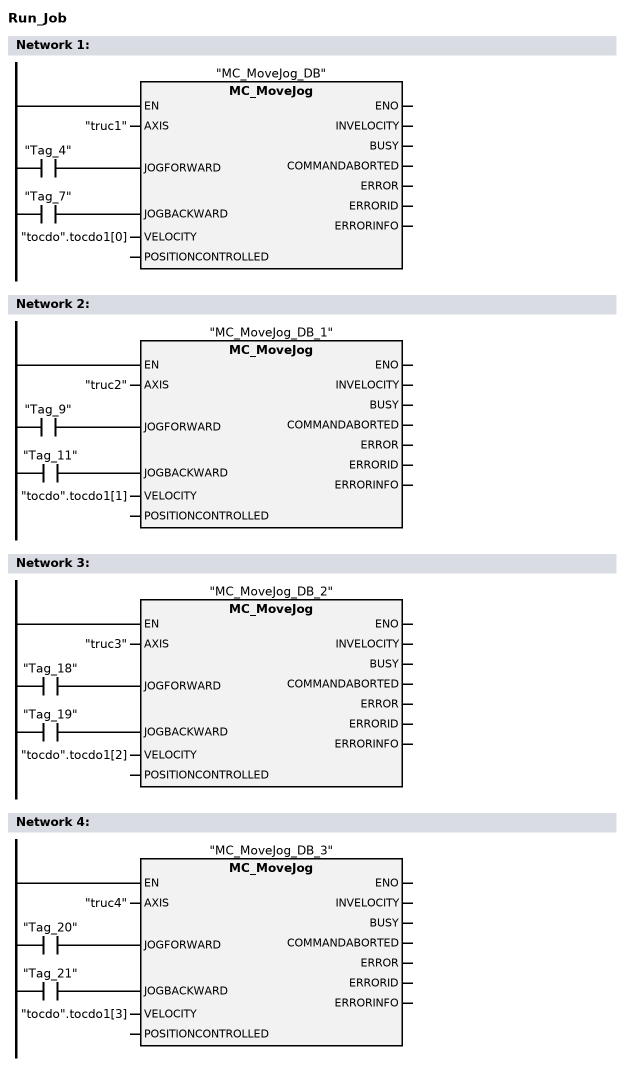
   "MC_MoveJog_DB"(Axis := "truc1",   // MC_MoveJog
                   JogForward := "Tag_4",
                   JogBackward := "Tag_7",
                   Velocity := "tocdo".tocdo1[0]);
END_REGION

REGION Network 2
   "MC_MoveJog_DB_1"(Axis := "truc2",   // MC_MoveJog
                     JogForward := "Tag_9",
                     JogBackward := "Tag_11",
                     Velocity := "tocdo".tocdo1[1]);
END_REGION

REGION Network 3
   "MC_MoveJog_DB_2"(Axis := "truc3",   // MC_MoveJog
                     JogForward := "Tag_18",
                     JogBackward := "Tag_19",
                     Velocity := "tocdo".tocdo1[2]);
END_REGION

REGION Network 4
   "MC_MoveJog_DB_3"(Axis := "truc4",   // MC_MoveJog
                     JogForward := "Tag_20",
                     JogBackward := "Tag_21",
                     Velocity := "tocdo".tocdo1[3]);
END_REGION
END_FUNCTION

FUNCTION "BT_Giua_Khau1" : Void   // FC5, LAD
{ S7_Optimized_Access := 'TRUE' }
VERSION : 0.1
BEGIN

REGION Network 1
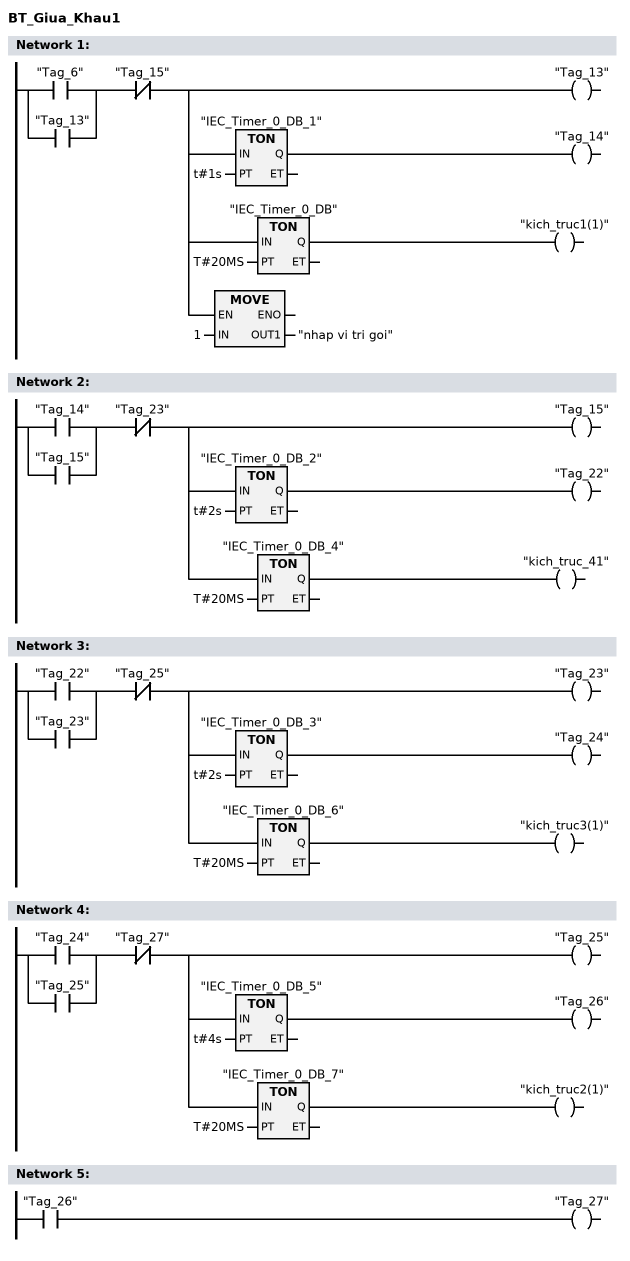
   "Tag_13" := ("Tag_6" OR "Tag_13") AND NOT "Tag_15";
   "IEC_Timer_0_DB_1".TON(IN := "Tag_13", PT := t#1s);
   "Tag_14" := "IEC_Timer_0_DB_1".Q;
   "IEC_Timer_0_DB".TON(IN := "Tag_13", PT := T#20MS);
   "kich_truc1(1)" := "IEC_Timer_0_DB".Q;
   IF "Tag_13" THEN "nhap vi tri goi" := 1; END_IF;
END_REGION

REGION Network 2
   "Tag_15" := ("Tag_14" OR "Tag_15") AND NOT "Tag_23";
   "IEC_Timer_0_DB_2".TON(IN := "Tag_15", PT := t#2s);
   "Tag_22" := "IEC_Timer_0_DB_2".Q;
   "IEC_Timer_0_DB_4".TON(IN := "Tag_15", PT := T#20MS);
   "kich_truc_41" := "IEC_Timer_0_DB_4".Q;
END_REGION

REGION Network 3
   "Tag_23" := ("Tag_22" OR "Tag_23") AND NOT "Tag_25";
   "IEC_Timer_0_DB_3".TON(IN := "Tag_23", PT := t#2s);
   "Tag_24" := "IEC_Timer_0_DB_3".Q;
   "IEC_Timer_0_DB_6".TON(IN := "Tag_23", PT := T#20MS);
   "kich_truc3(1)" := "IEC_Timer_0_DB_6".Q;
END_REGION

REGION Network 4
   "Tag_25" := ("Tag_24" OR "Tag_25") AND NOT "Tag_27";
   "IEC_Timer_0_DB_5".TON(IN := "Tag_25", PT := t#4s);
   "Tag_26" := "IEC_Timer_0_DB_5".Q;
   "IEC_Timer_0_DB_7".TON(IN := "Tag_25", PT := T#20MS);
   "kich_truc2(1)" := "IEC_Timer_0_DB_7".Q;
END_REGION

REGION Network 5
   RUNG wire#powerrail
      Contact( "Tag_26" )
      Coil( "Tag_27" )
   END_RUNG
   // the same network as SCL:
   "Tag_27" := "Tag_26";
END_REGION
END_FUNCTION

FUNCTION "BT_Giua_Khau2" : Void   // FC6, LAD
{ S7_Optimized_Access := 'TRUE' }
VERSION : 0.1
BEGIN

REGION Network 1
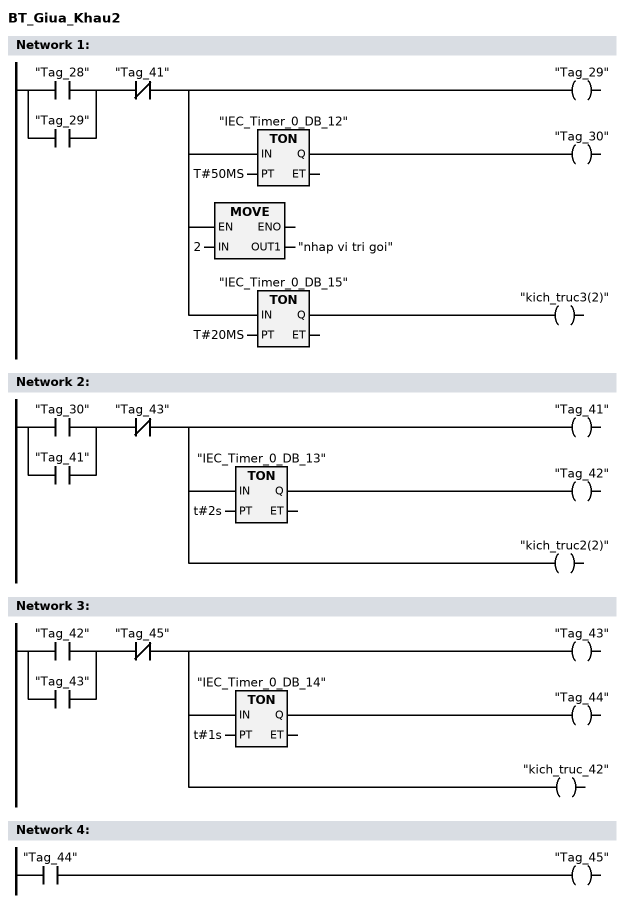
   "Tag_29" := ("Tag_28" OR "Tag_29") AND NOT "Tag_41";
   "IEC_Timer_0_DB_12".TON(IN := "Tag_29", PT := T#50MS);
   "Tag_30" := "IEC_Timer_0_DB_12".Q;
   IF "Tag_29" THEN "nhap vi tri goi" := 2; END_IF;
   "IEC_Timer_0_DB_15".TON(IN := "Tag_29", PT := T#20MS);
   "kich_truc3(2)" := "IEC_Timer_0_DB_15".Q;
END_REGION

REGION Network 2
   "Tag_41" := ("Tag_30" OR "Tag_41") AND NOT "Tag_43";
   "IEC_Timer_0_DB_13".TON(IN := "Tag_41", PT := t#2s);
   "Tag_42" := "IEC_Timer_0_DB_13".Q;
   "kich_truc2(2)" := "Tag_41";
END_REGION

REGION Network 3
   "Tag_43" := ("Tag_42" OR "Tag_43") AND NOT "Tag_45";
   "IEC_Timer_0_DB_14".TON(IN := "Tag_43", PT := t#1s);
   "Tag_44" := "IEC_Timer_0_DB_14".Q;
   "kich_truc_42" := "Tag_43";
END_REGION

REGION Network 4
   RUNG wire#powerrail
      Contact( "Tag_44" )
      Coil( "Tag_45" )
   END_RUNG
   // the same network as SCL:
   "Tag_45" := "Tag_44";
END_REGION
END_FUNCTION

FUNCTION "BT_Giua_khau3" : Void   // FC7, LAD
{ S7_Optimized_Access := 'TRUE' }
VERSION : 0.1
BEGIN

REGION Network 1
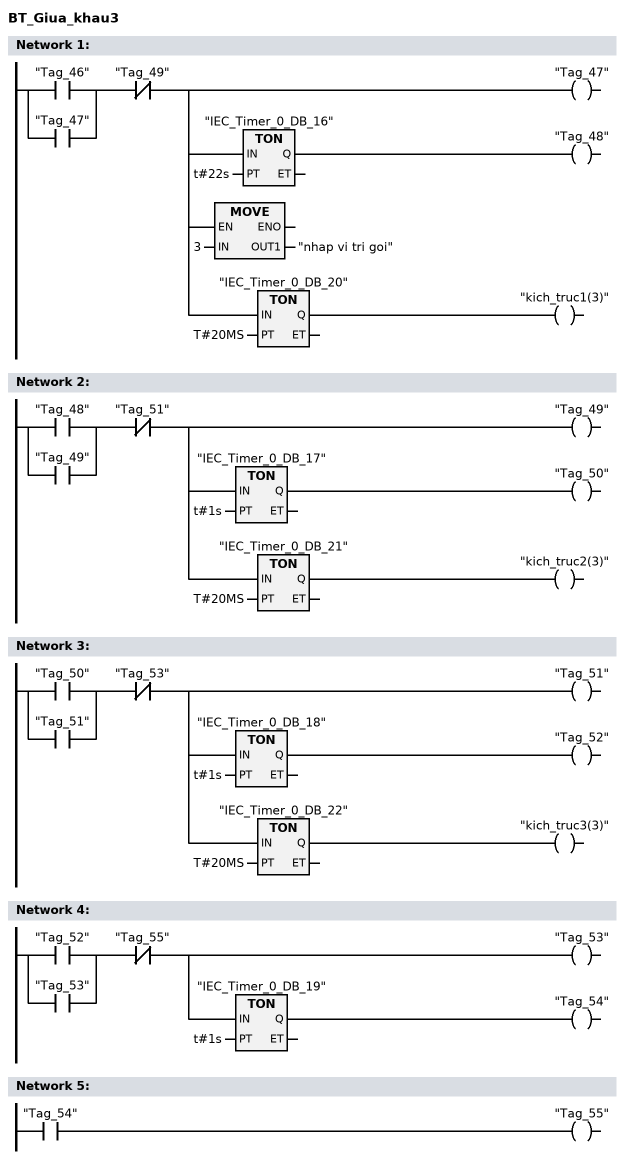
   "Tag_47" := ("Tag_46" OR "Tag_47") AND NOT "Tag_49";
   "IEC_Timer_0_DB_16".TON(IN := "Tag_47", PT := t#22s);
   "Tag_48" := "IEC_Timer_0_DB_16".Q;
   IF "Tag_47" THEN "nhap vi tri goi" := 3; END_IF;
   "IEC_Timer_0_DB_20".TON(IN := "Tag_47", PT := T#20MS);
   "kich_truc1(3)" := "IEC_Timer_0_DB_20".Q;
END_REGION

REGION Network 2
   "Tag_49" := ("Tag_48" OR "Tag_49") AND NOT "Tag_51";
   "IEC_Timer_0_DB_17".TON(IN := "Tag_49", PT := t#1s);
   "Tag_50" := "IEC_Timer_0_DB_17".Q;
   "IEC_Timer_0_DB_21".TON(IN := "Tag_49", PT := T#20MS);
   "kich_truc2(3)" := "IEC_Timer_0_DB_21".Q;
END_REGION

REGION Network 3
   "Tag_51" := ("Tag_50" OR "Tag_51") AND NOT "Tag_53";
   "IEC_Timer_0_DB_18".TON(IN := "Tag_51", PT := t#1s);
   "Tag_52" := "IEC_Timer_0_DB_18".Q;
   "IEC_Timer_0_DB_22".TON(IN := "Tag_51", PT := T#20MS);
   "kich_truc3(3)" := "IEC_Timer_0_DB_22".Q;
END_REGION

REGION Network 4
   "Tag_53" := ("Tag_52" OR "Tag_53") AND NOT "Tag_55";
   "IEC_Timer_0_DB_19".TON(IN := "Tag_53", PT := t#1s);
   "Tag_54" := "IEC_Timer_0_DB_19".Q;
END_REGION

REGION Network 5
   RUNG wire#powerrail
      Contact( "Tag_54" )
      Coil( "Tag_55" )
   END_RUNG
   // the same network as SCL:
   "Tag_55" := "Tag_54";
END_REGION
END_FUNCTION

FUNCTION "ve_Homing" : Void   // FC8, LAD
{ S7_Optimized_Access := 'TRUE' }
VERSION : 0.1
BEGIN

REGION Network 1
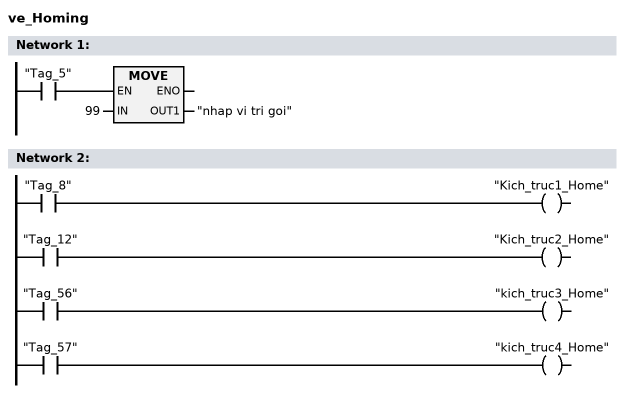
   RUNG wire#powerrail
      Contact( "Tag_5" )
      Move(in := 99, out1 => "nhap vi tri goi")
   END_RUNG
   // the same network as SCL:
   IF "Tag_5" THEN "nhap vi tri goi" := 99; END_IF;
END_REGION

REGION Network 2
   RUNG wire#powerrail
      Contact( "Tag_8" )
      Coil( "Kich_truc1_Home" )
   END_RUNG
   RUNG wire#powerrail
      Contact( "Tag_12" )
      Coil( "Kich_truc2_Home" )
   END_RUNG
   RUNG wire#powerrail
      Contact( "Tag_56" )
      Coil( "kich_truc3_Home" )
   END_RUNG
   RUNG wire#powerrail
      Contact( "Tag_57" )
      Coil( "kich_truc4_Home" )
   END_RUNG
   // the same network as SCL:
   "Kich_truc1_Home" := "Tag_8";
   "Kich_truc2_Home" := "Tag_12";
   "kich_truc3_Home" := "Tag_56";
   "kich_truc4_Home" := "Tag_57";
END_REGION
END_FUNCTION

FUNCTION "chuyen_dong_BT_Giua" : Void   // FC9, LAD
{ S7_Optimized_Access := 'TRUE' }
VERSION : 0.1
BEGIN

REGION Network 1
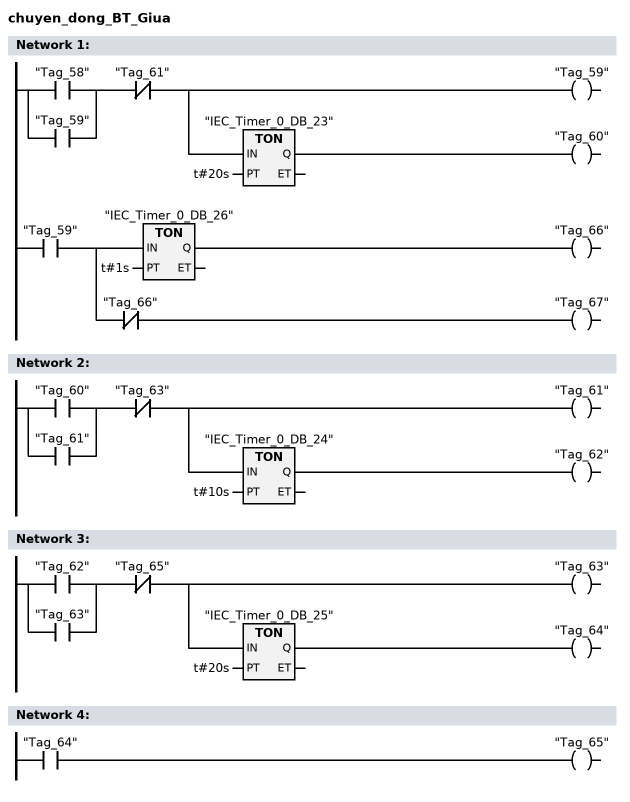
   "Tag_59" := ("Tag_58" OR "Tag_59") AND NOT "Tag_61";
   "IEC_Timer_0_DB_23".TON(IN := "Tag_59", PT := t#20s);
   "Tag_60" := "IEC_Timer_0_DB_23".Q;
   "IEC_Timer_0_DB_26".TON(IN := "Tag_59", PT := t#1s);
   "Tag_66" := "IEC_Timer_0_DB_26".Q;
   "Tag_67" := "Tag_59" AND NOT "Tag_66";
END_REGION

REGION Network 2
   "Tag_61" := ("Tag_60" OR "Tag_61") AND NOT "Tag_63";
   "IEC_Timer_0_DB_24".TON(IN := "Tag_61", PT := t#10s);
   "Tag_62" := "IEC_Timer_0_DB_24".Q;
END_REGION

REGION Network 3
   "Tag_63" := ("Tag_62" OR "Tag_63") AND NOT "Tag_65";
   "IEC_Timer_0_DB_25".TON(IN := "Tag_63", PT := t#20s);
   "Tag_64" := "IEC_Timer_0_DB_25".Q;
END_REGION

REGION Network 4
   RUNG wire#powerrail
      Contact( "Tag_64" )
      Coil( "Tag_65" )
   END_RUNG
   // the same network as SCL:
   "Tag_65" := "Tag_64";
END_REGION
END_FUNCTION

ORGANIZATION_BLOCK "Main"   // OB1, LAD, ProgramCycle
TITLE = "Main Program Sweep (Cycle)"
{ S7_Optimized_Access := 'TRUE' }
VERSION : 0.1
   VAR_INPUT
      Initial_Call : Bool;   // Initial call of this OB
      Remanence : Bool;   // =True, if remanent data are available
   END_VAR
BEGIN

REGION Network 1
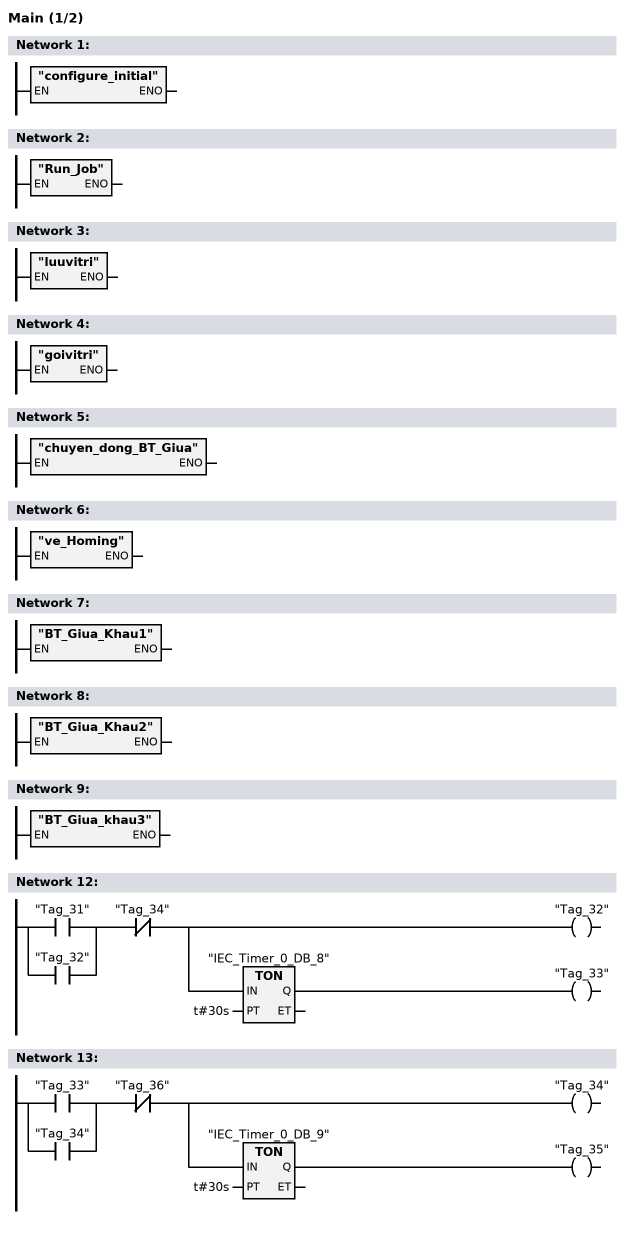
   RUNG wire#powerrail
      "configure_initial"()
   END_RUNG
   // the same network as SCL:
   "configure_initial"();
END_REGION

REGION Network 2
   RUNG wire#powerrail
      "Run_Job"()
   END_RUNG
   // the same network as SCL:
   "Run_Job"();
END_REGION

REGION Network 3
   RUNG wire#powerrail
      "luuvitri"()
   END_RUNG
   // the same network as SCL:
   "luuvitri"();
END_REGION

REGION Network 4
   RUNG wire#powerrail
      "goivitri"()
   END_RUNG
   // the same network as SCL:
   "goivitri"();
END_REGION

REGION Network 5
   RUNG wire#powerrail
      "chuyen_dong_BT_Giua"()
   END_RUNG
   // the same network as SCL:
   "chuyen_dong_BT_Giua"();
END_REGION

REGION Network 6
   RUNG wire#powerrail
      "ve_Homing"()
   END_RUNG
   // the same network as SCL:
   "ve_Homing"();
END_REGION

REGION Network 7
   RUNG wire#powerrail
      "BT_Giua_Khau1"()
   END_RUNG
   // the same network as SCL:
   "BT_Giua_Khau1"();
END_REGION

REGION Network 8
   RUNG wire#powerrail
      "BT_Giua_Khau2"()
   END_RUNG
   // the same network as SCL:
   "BT_Giua_Khau2"();
END_REGION

REGION Network 9
   RUNG wire#powerrail
      "BT_Giua_khau3"()
   END_RUNG
   // the same network as SCL:
   "BT_Giua_khau3"();
END_REGION

REGION Network 12
   "Tag_32" := ("Tag_31" OR "Tag_32") AND NOT "Tag_34";
   "IEC_Timer_0_DB_8".TON(IN := "Tag_32", PT := t#30s);
   "Tag_33" := "IEC_Timer_0_DB_8".Q;
END_REGION

REGION Network 13
   "Tag_34" := ("Tag_33" OR "Tag_34") AND NOT "Tag_36";
   "IEC_Timer_0_DB_9".TON(IN := "Tag_34", PT := t#30s);
   "Tag_35" := "IEC_Timer_0_DB_9".Q;
END_REGION

REGION Network 14
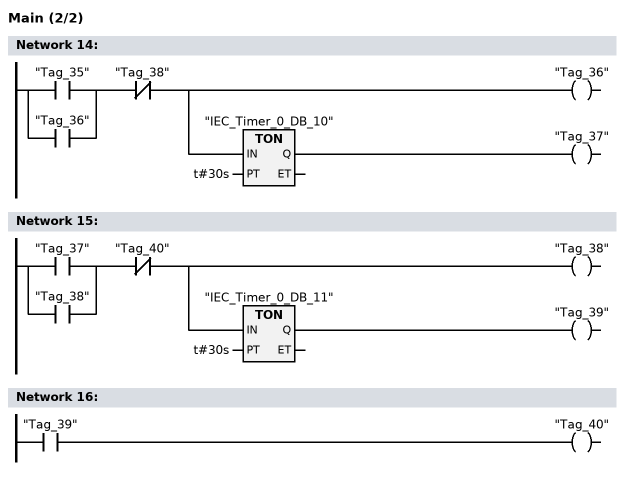
   "Tag_36" := ("Tag_35" OR "Tag_36") AND NOT "Tag_38";
   "IEC_Timer_0_DB_10".TON(IN := "Tag_36", PT := t#30s);
   "Tag_37" := "IEC_Timer_0_DB_10".Q;
END_REGION

REGION Network 15
   "Tag_38" := ("Tag_37" OR "Tag_38") AND NOT "Tag_40";
   "IEC_Timer_0_DB_11".TON(IN := "Tag_38", PT := t#30s);
   "Tag_39" := "IEC_Timer_0_DB_11".Q;
END_REGION

REGION Network 16
   RUNG wire#powerrail
      Contact( "Tag_39" )
      Coil( "Tag_40" )
   END_RUNG
   // the same network as SCL:
   "Tag_40" := "Tag_39";
END_REGION
END_ORGANIZATION_BLOCK